// TIA Portal V16 export
// export: Created 2022-11-14T17:35:26.3349188Z, ExportSetting WithDefaults, DisplayName Totally Integrated Automation Portal, DisplayVersion V16, DisplayName TIA Portal Version Control Interface, DisplayVersion V16, DisplayName TIA Portal Openness, DisplayVersion V16, DisplayName STEP 7 Professional, DisplayVersion V16, DisplayName STEP 7 Safety, DisplayVersion V16, DisplayName WinCC Advanced, DisplayVersion V16
FUNCTION "FC32_ConveyorInverter_REV" : Void   // FC32, LAD
TITLE = Conveyor management with inverter
{ S7_Optimized_Access := 'FALSE' }
AUTHOR : Robopac
VERSION : 0.0
// stored: AutoNumber false, IsIECCheckEnabled false, SetENOAutomatically false, UDAEnableTagReadback false
   VAR_TEMP
      TimeUpwardTableCycle : Word;
      TimeUpwardTableCycleInt : Int;
      TempWord : Word;
   END_VAR
   VAR_TEMP   // added for the SCL form of the ladder/FBD networks
      _w1 : Bool;
   END_VAR
BEGIN

REGION Network 1: Timer SA type for conveyor motor
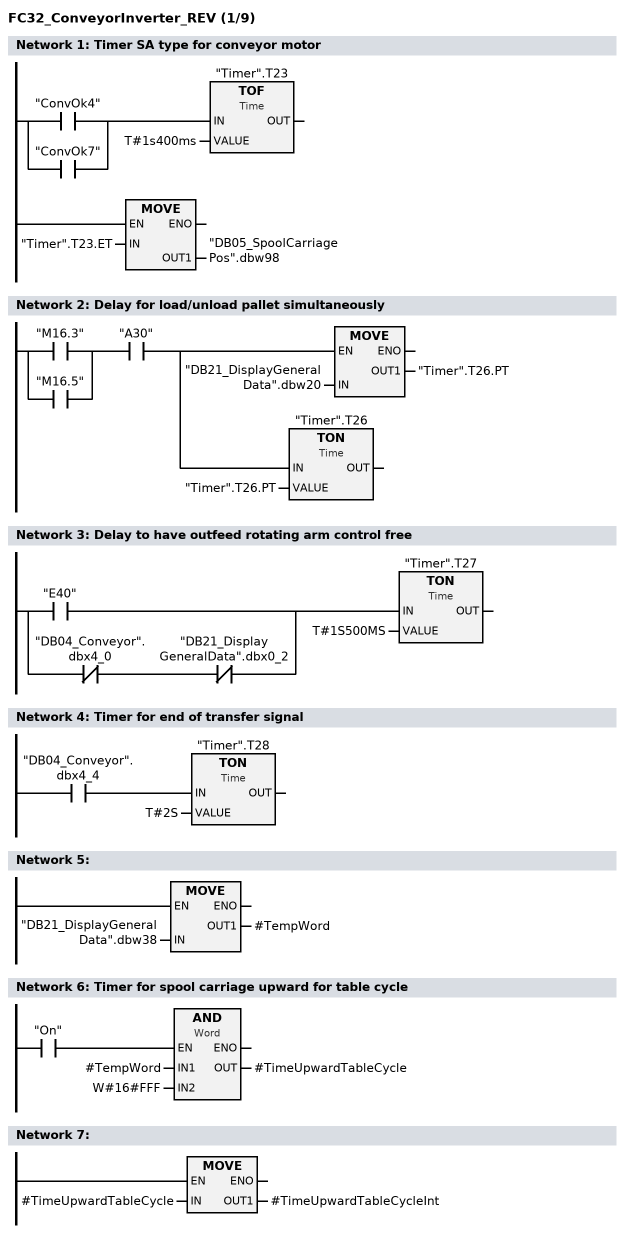
   "Timer".T23.TOF(IN := "ConvOk4" OR "ConvOk7", PT := T#1s400ms);   // TOF coil
   "DB05_SpoolCarriagePos".dbw98 := "Timer".T23.ET;
END_REGION

REGION Network 2: Delay for load/unload pallet simultaneously
   #_w1 := ("M16.3" OR "M16.5") AND "A30";
   IF #_w1 THEN "Timer".T26.PT := "DB21_DisplayGeneralData".dbw20; END_IF;
   "Timer".T26.TON(IN := #_w1, PT := "Timer".T26.PT);   // TON coil
END_REGION

REGION Network 3: Delay to have outfeed rotating arm control free
   "Timer".T27.TON(IN := "E40" OR (NOT "DB04_Conveyor".dbx4_0 AND NOT "DB21_DisplayGeneralData".dbx0_2), PT := T#1S500MS);   // TON coil
END_REGION

REGION Network 4: Timer for end of transfer signal
   "Timer".T28.TON(IN := "DB04_Conveyor".dbx4_4, PT := T#2S);   // TON coil
END_REGION

REGION Network 5
   RUNG wire#powerrail
      { S7_GenerateENO := "TRUE" } Move(in := "DB21_DisplayGeneralData".dbw38, out1 => #TempWord)
   END_RUNG
   // the same network as SCL:
   #TempWord := "DB21_DisplayGeneralData".dbw38;
END_REGION

REGION Network 6: Timer for spool carriage upward for table cycle
   RUNG wire#powerrail
      Contact( "On" )
      { S7_Templates := "SrcType := Word"; S7_GenerateENO := "TRUE" } And(in1 := #TempWord, in2 := W#16#FFF, out => #TimeUpwardTableCycle)
   END_RUNG
   // the same network as SCL:
   IF "On" THEN #TimeUpwardTableCycle := #TempWord AND W#16#FFF; END_IF;
END_REGION

REGION Network 7
   RUNG wire#powerrail
      { S7_GenerateENO := "TRUE" } Move(in := #TimeUpwardTableCycle, out1 => #TimeUpwardTableCycleInt)
   END_RUNG
   // the same network as SCL:
   #TimeUpwardTableCycleInt := #TimeUpwardTableCycle;
END_REGION

REGION Network 8: Timer for spool carriage upward for table cycle
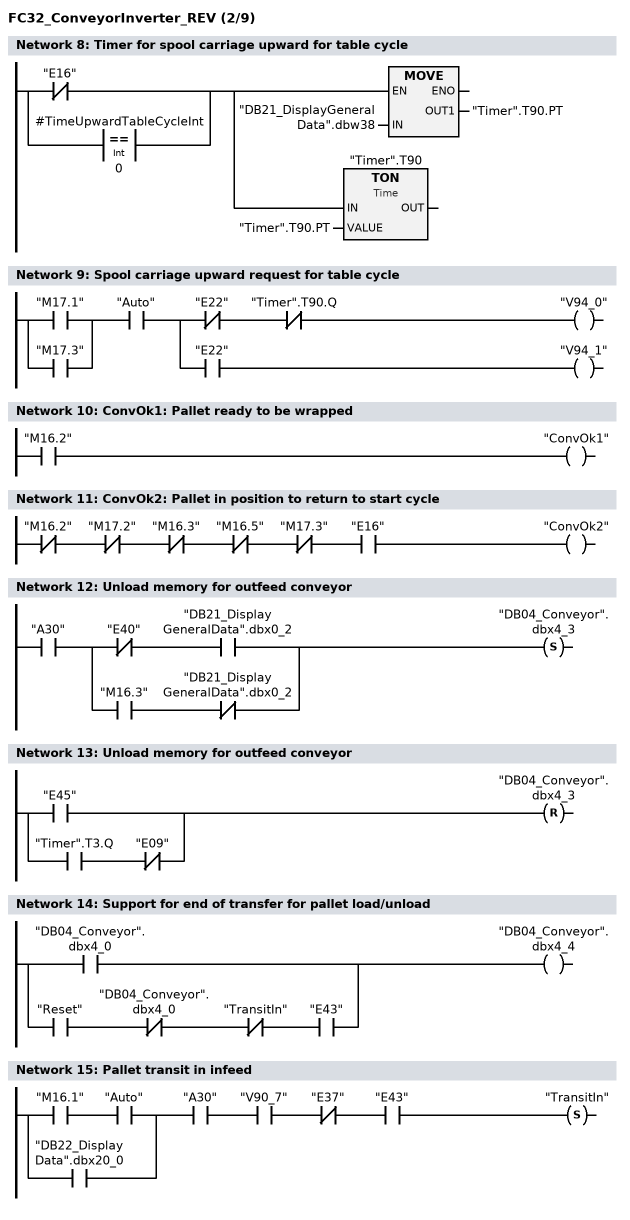
   #_w1 := NOT "E16" OR (#TimeUpwardTableCycleInt = 0);
   IF #_w1 THEN "Timer".T90.PT := "DB21_DisplayGeneralData".dbw38; END_IF;
   "Timer".T90.TON(IN := #_w1, PT := "Timer".T90.PT);   // TON coil
END_REGION

REGION Network 9: Spool carriage upward request for table cycle
   RUNG wire#powerrail
      Contact( "M17.1" )
      wire#w1
      Contact( "Auto" )
      wire#w2
      I_Contact( "E22" )
      I_Contact( "Timer".T90.Q )
      Coil( "V94_0" )
   END_RUNG
   RUNG wire#powerrail
      Contact( "M17.3" )
   END_RUNG wire#w1
   RUNG wire#w2
      Contact( "E22" )
      Coil( "V94_1" )
   END_RUNG
   // the same network as SCL:
   #_w1 := ("M17.1" OR "M17.3") AND "Auto";
   "V94_0" := #_w1 AND NOT "E22" AND NOT "Timer".T90.Q;
   "V94_1" := #_w1 AND "E22";
END_REGION

REGION Network 10: ConvOk1: Pallet ready to be wrapped
   RUNG wire#powerrail
      Contact( "M16.2" )
      Coil( "ConvOk1" )
   END_RUNG
   // the same network as SCL:
   "ConvOk1" := "M16.2";
END_REGION

REGION Network 11: ConvOk2: Pallet in position to return to start cycle
   RUNG wire#powerrail
      I_Contact( "M16.2" )
      I_Contact( "M17.2" )
      I_Contact( "M16.3" )
      I_Contact( "M16.5" )
      I_Contact( "M17.3" )
      Contact( "E16" )
      Coil( "ConvOk2" )
   END_RUNG
   // the same network as SCL:
   "ConvOk2" := NOT "M16.2" AND NOT "M17.2" AND NOT "M16.3" AND NOT "M16.5" AND NOT "M17.3" AND "E16";
END_REGION

REGION Network 12: Unload memory for outfeed conveyor
   RUNG wire#powerrail
      Contact( "A30" )
      wire#w1
      I_Contact( "E40" )
      Contact( "DB21_DisplayGeneralData".dbx0_2 )
      wire#w2
      S_Coil( "DB04_Conveyor".dbx4_3 )
   END_RUNG
   RUNG wire#w1
      Contact( "M16.3" )
      I_Contact( "DB21_DisplayGeneralData".dbx0_2 )
   END_RUNG wire#w2
   // the same network as SCL:
   IF "A30" AND ((NOT "E40" AND "DB21_DisplayGeneralData".dbx0_2) OR ("M16.3" AND NOT "DB21_DisplayGeneralData".dbx0_2)) THEN
       "DB04_Conveyor".dbx4_3 := TRUE;
   END_IF;
END_REGION

REGION Network 13: Unload memory for outfeed conveyor
   RUNG wire#powerrail
      Contact( "E45" )
      wire#w1
      R_Coil( "DB04_Conveyor".dbx4_3 )
   END_RUNG
   RUNG wire#powerrail
      Contact( "Timer".T3.Q )
      I_Contact( "E09" )
   END_RUNG wire#w1
   // the same network as SCL:
   IF "E45" OR ("Timer".T3.Q AND NOT "E09") THEN "DB04_Conveyor".dbx4_3 := FALSE; END_IF;
END_REGION

REGION Network 14: Support for end of transfer for pallet load/unload
   RUNG wire#powerrail
      Contact( "DB04_Conveyor".dbx4_0 )
      wire#w1
      Coil( "DB04_Conveyor".dbx4_4 )
   END_RUNG
   RUNG wire#powerrail
      Contact( "Reset" )
      I_Contact( "DB04_Conveyor".dbx4_0 )
      I_Contact( "TransitIn" )
      Contact( "E43" )
   END_RUNG wire#w1
   // the same network as SCL:
   "DB04_Conveyor".dbx4_4 := "DB04_Conveyor".dbx4_0 OR ("Reset" AND NOT "DB04_Conveyor".dbx4_0 AND NOT "TransitIn" AND "E43");
END_REGION

REGION Network 15: Pallet transit in infeed
   RUNG wire#powerrail
      Contact( "M16.1" )
      Contact( "Auto" )
      wire#w1
      Contact( "A30" )
      Contact( "V90_7" )
      I_Contact( "E37" )
      Contact( "E43" )
      S_Coil( "TransitIn" )
   END_RUNG
   RUNG wire#powerrail
      Contact( "DB22_DisplayData".dbx20_0 )
   END_RUNG wire#w1
   // the same network as SCL:
   IF (("M16.1" AND "Auto") OR "DB22_DisplayData".dbx20_0) AND "A30" AND "V90_7" AND NOT "E37" AND "E43" THEN
       "TransitIn" := TRUE;
   END_IF;
END_REGION

REGION Network 16: Pallet transit in infeed
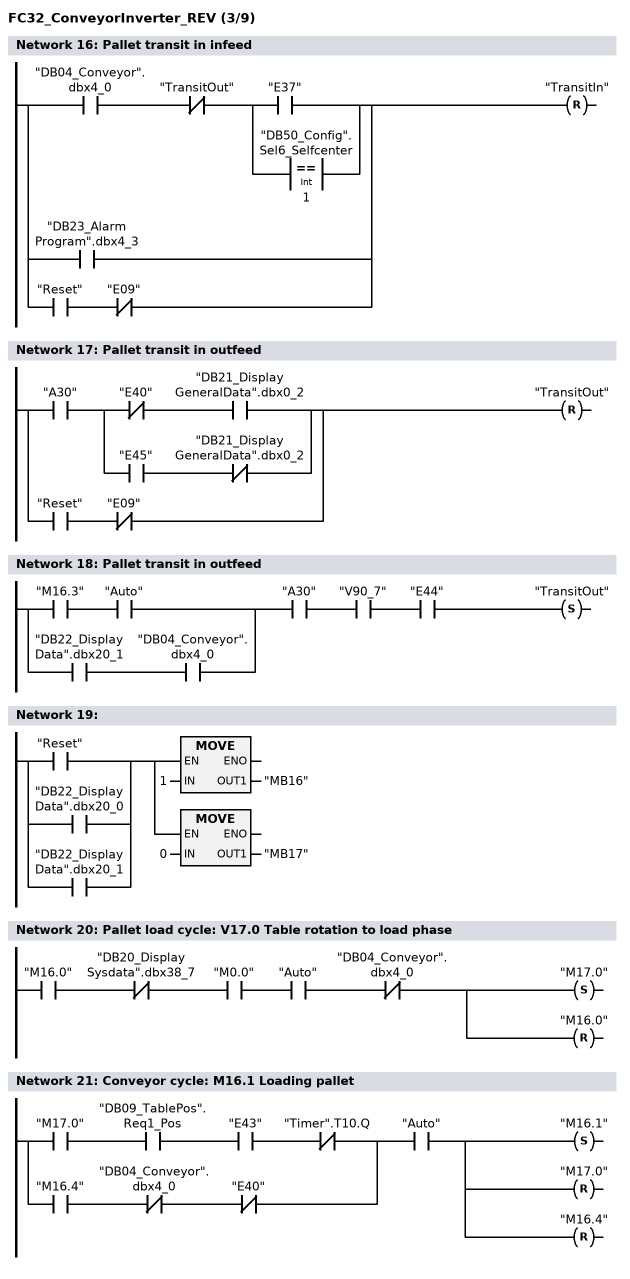
   IF ("DB04_Conveyor".dbx4_0 AND NOT "TransitOut" AND (("DB50_Config".Sel6_Selfcenter = 1) OR "E37")) OR "DB23_AlarmProgram".dbx4_3 OR ("Reset" AND NOT "E09") THEN
       "TransitIn" := FALSE;
   END_IF;
END_REGION

REGION Network 17: Pallet transit in outfeed
   RUNG wire#powerrail
      Contact( "A30" )
      wire#w1
      I_Contact( "E40" )
      Contact( "DB21_DisplayGeneralData".dbx0_2 )
      wire#w2
      R_Coil( "TransitOut" )
   END_RUNG
   RUNG wire#w1
      Contact( "E45" )
      I_Contact( "DB21_DisplayGeneralData".dbx0_2 )
   END_RUNG wire#w2
   RUNG wire#powerrail
      Contact( "Reset" )
      I_Contact( "E09" )
   END_RUNG wire#w2
   // the same network as SCL:
   IF ("A30" AND ((NOT "E40" AND "DB21_DisplayGeneralData".dbx0_2) OR ("E45" AND NOT "DB21_DisplayGeneralData".dbx0_2))) OR ("Reset" AND NOT "E09") THEN
       "TransitOut" := FALSE;
   END_IF;
END_REGION

REGION Network 18: Pallet transit in outfeed
   RUNG wire#powerrail
      Contact( "M16.3" )
      Contact( "Auto" )
      wire#w1
      Contact( "A30" )
      Contact( "V90_7" )
      Contact( "E44" )
      S_Coil( "TransitOut" )
   END_RUNG
   RUNG wire#powerrail
      Contact( "DB22_DisplayData".dbx20_1 )
      Contact( "DB04_Conveyor".dbx4_0 )
   END_RUNG wire#w1
   // the same network as SCL:
   IF (("M16.3" AND "Auto") OR ("DB22_DisplayData".dbx20_1 AND "DB04_Conveyor".dbx4_0)) AND "A30" AND "V90_7" AND "E44" THEN
       "TransitOut" := TRUE;
   END_IF;
END_REGION

REGION Network 19
   RUNG wire#powerrail
      Contact( "Reset" )
      wire#w1
      { S7_GenerateENO := "TRUE" } Move(in := 1, out1 => "MB16")
   END_RUNG
   RUNG wire#powerrail
      Contact( "DB22_DisplayData".dbx20_0 )
   END_RUNG wire#w1
   RUNG wire#powerrail
      Contact( "DB22_DisplayData".dbx20_1 )
   END_RUNG wire#w1
   RUNG wire#w1
      { S7_GenerateENO := "TRUE" } Move(in := 0, out1 => "MB17")
   END_RUNG
   // the same network as SCL:
   IF "Reset" OR "DB22_DisplayData".dbx20_0 OR "DB22_DisplayData".dbx20_1 THEN
       "MB16" := 1;
       "MB17" := 0;
   END_IF;
END_REGION

REGION Network 20: Pallet load cycle: V17.0 Table rotation to load phase
   RUNG wire#powerrail
      Contact( "M16.0" )
      I_Contact( "DB20_DisplaySysdata".dbx38_7 )
      Contact( "M0.0" )
      Contact( "Auto" )
      I_Contact( "DB04_Conveyor".dbx4_0 )
      wire#w1
      S_Coil( "M17.0" )
   END_RUNG
   RUNG wire#w1
      R_Coil( "M16.0" )
   END_RUNG
   // the same network as SCL:
   IF "M16.0" AND NOT "DB20_DisplaySysdata".dbx38_7 AND "M0.0" AND "Auto" AND NOT "DB04_Conveyor".dbx4_0 THEN
       "M17.0" := TRUE;
       "M16.0" := FALSE;
   END_IF;
END_REGION

REGION Network 21: Conveyor cycle: M16.1 Loading pallet
   RUNG wire#powerrail
      Contact( "M17.0" )
      Contact( "DB09_TablePos".Req1_Pos )
      Contact( "E43" )
      I_Contact( "Timer".T10.Q )
      wire#w1
      Contact( "Auto" )
      wire#w2
      S_Coil( "M16.1" )
   END_RUNG
   RUNG wire#powerrail
      Contact( "M16.4" )
      I_Contact( "DB04_Conveyor".dbx4_0 )
      I_Contact( "E40" )
   END_RUNG wire#w1
   RUNG wire#w2
      R_Coil( "M17.0" )
   END_RUNG
   RUNG wire#w2
      R_Coil( "M16.4" )
   END_RUNG
   // the same network as SCL:
   IF (("M17.0" AND "DB09_TablePos".Req1_Pos AND "E43" AND NOT "Timer".T10.Q) OR ("M16.4" AND NOT "DB04_Conveyor".dbx4_0 AND NOT "E40")) AND "Auto" THEN
       "M16.1" := TRUE;
   END_IF;
   #_w1 := (("M17.0" AND "DB09_TablePos".Req1_Pos AND "E43" AND NOT "Timer".T10.Q) OR ("M16.4" AND NOT "DB04_Conveyor".dbx4_0 AND NOT "E40")) AND "Auto";
   IF #_w1 THEN
       "M17.0" := FALSE;
       "M16.4" := FALSE;
   END_IF;
END_REGION

REGION Network 22: Pallet load cycle: V17.1 Table rotation to machine phase from lo
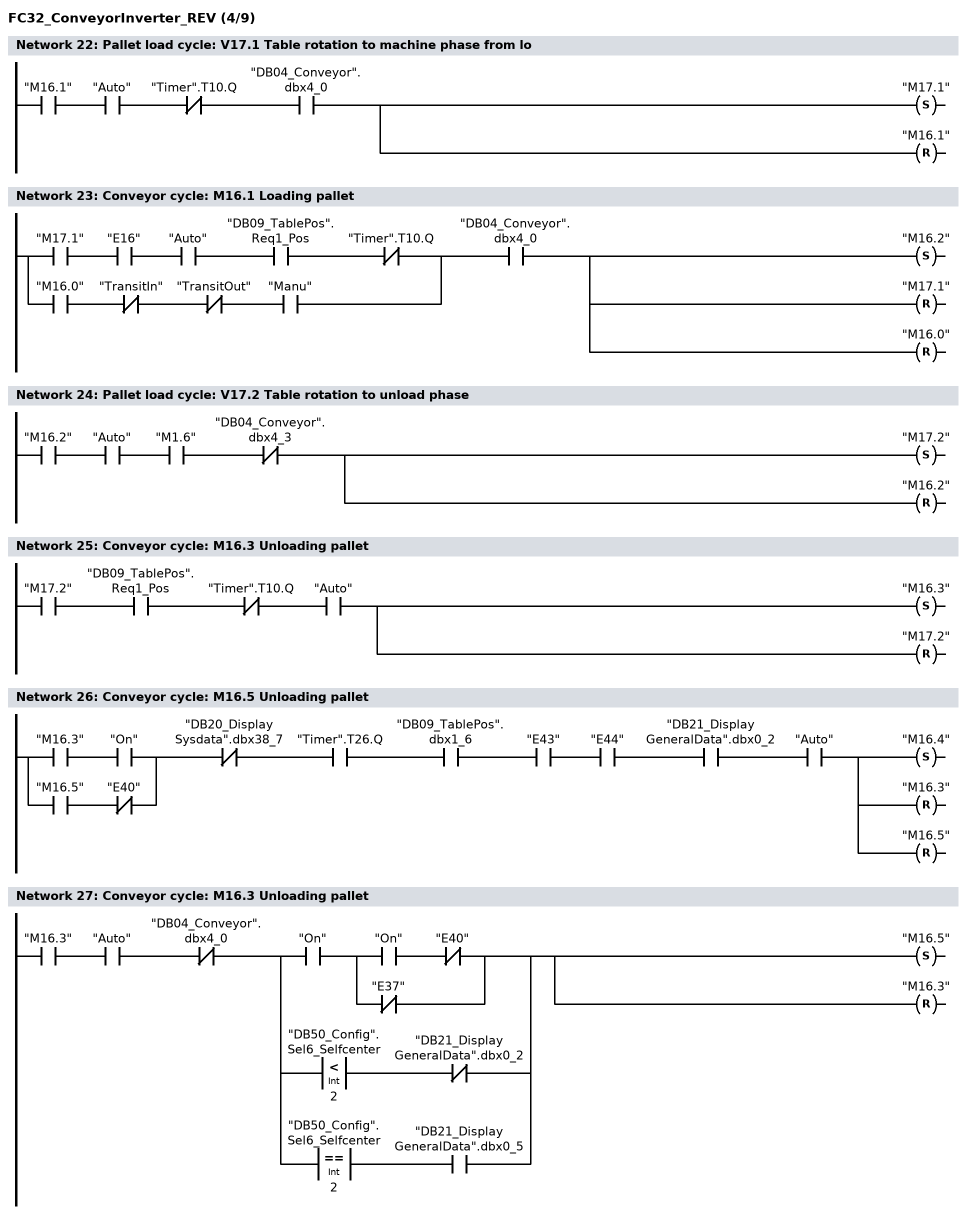
   RUNG wire#powerrail
      Contact( "M16.1" )
      Contact( "Auto" )
      I_Contact( "Timer".T10.Q )
      Contact( "DB04_Conveyor".dbx4_0 )
      wire#w1
      S_Coil( "M17.1" )
   END_RUNG
   RUNG wire#w1
      R_Coil( "M16.1" )
   END_RUNG
   // the same network as SCL:
   IF "M16.1" AND "Auto" AND NOT "Timer".T10.Q AND "DB04_Conveyor".dbx4_0 THEN
       "M17.1" := TRUE;
       "M16.1" := FALSE;
   END_IF;
END_REGION

REGION Network 23: Conveyor cycle: M16.1 Loading pallet
   RUNG wire#powerrail
      Contact( "M17.1" )
      Contact( "E16" )
      Contact( "Auto" )
      Contact( "DB09_TablePos".Req1_Pos )
      I_Contact( "Timer".T10.Q )
      wire#w1
      Contact( "DB04_Conveyor".dbx4_0 )
      wire#w2
      S_Coil( "M16.2" )
   END_RUNG
   RUNG wire#powerrail
      Contact( "M16.0" )
      I_Contact( "TransitIn" )
      I_Contact( "TransitOut" )
      Contact( "Manu" )
   END_RUNG wire#w1
   RUNG wire#w2
      R_Coil( "M17.1" )
   END_RUNG
   RUNG wire#w2
      R_Coil( "M16.0" )
   END_RUNG
   // the same network as SCL:
   IF (("M17.1" AND "E16" AND "Auto" AND "DB09_TablePos".Req1_Pos AND NOT "Timer".T10.Q) OR ("M16.0" AND NOT "TransitIn" AND NOT "TransitOut" AND "Manu")) AND "DB04_Conveyor".dbx4_0 THEN
       "M16.2" := TRUE;
   END_IF;
   #_w1 := (("M17.1" AND "E16" AND "Auto" AND "DB09_TablePos".Req1_Pos AND NOT "Timer".T10.Q) OR ("M16.0" AND NOT "TransitIn" AND NOT "TransitOut" AND "Manu")) AND "DB04_Conveyor".dbx4_0;
   IF #_w1 THEN
       "M17.1" := FALSE;
       "M16.0" := FALSE;
   END_IF;
END_REGION

REGION Network 24: Pallet load cycle: V17.2 Table rotation to unload phase
   RUNG wire#powerrail
      Contact( "M16.2" )
      Contact( "Auto" )
      Contact( "M1.6" )
      I_Contact( "DB04_Conveyor".dbx4_3 )
      wire#w1
      S_Coil( "M17.2" )
   END_RUNG
   RUNG wire#w1
      R_Coil( "M16.2" )
   END_RUNG
   // the same network as SCL:
   IF "M16.2" AND "Auto" AND "M1.6" AND NOT "DB04_Conveyor".dbx4_3 THEN
       "M17.2" := TRUE;
       "M16.2" := FALSE;
   END_IF;
END_REGION

REGION Network 25: Conveyor cycle: M16.3 Unloading pallet
   RUNG wire#powerrail
      Contact( "M17.2" )
      Contact( "DB09_TablePos".Req1_Pos )
      I_Contact( "Timer".T10.Q )
      Contact( "Auto" )
      wire#w1
      S_Coil( "M16.3" )
   END_RUNG
   RUNG wire#w1
      R_Coil( "M17.2" )
   END_RUNG
   // the same network as SCL:
   IF "M17.2" AND "DB09_TablePos".Req1_Pos AND NOT "Timer".T10.Q AND "Auto" THEN
       "M16.3" := TRUE;
       "M17.2" := FALSE;
   END_IF;
END_REGION

REGION Network 26: Conveyor cycle: M16.5 Unloading pallet
   RUNG wire#powerrail
      Contact( "M16.3" )
      Contact( "On" )
      wire#w1
      I_Contact( "DB20_DisplaySysdata".dbx38_7 )
      Contact( "Timer".T26.Q )
      Contact( "DB09_TablePos".dbx1_6 )
      Contact( "E43" )
      Contact( "E44" )
      Contact( "DB21_DisplayGeneralData".dbx0_2 )
      Contact( "Auto" )
      wire#w2
      S_Coil( "M16.4" )
   END_RUNG
   RUNG wire#powerrail
      Contact( "M16.5" )
      I_Contact( "E40" )
   END_RUNG wire#w1
   RUNG wire#w2
      R_Coil( "M16.3" )
   END_RUNG
   RUNG wire#w2
      R_Coil( "M16.5" )
   END_RUNG
   // the same network as SCL:
   IF (("M16.3" AND "On") OR ("M16.5" AND NOT "E40")) AND NOT "DB20_DisplaySysdata".dbx38_7 AND "Timer".T26.Q AND "DB09_TablePos".dbx1_6 AND "E43" AND "E44" AND "DB21_DisplayGeneralData".dbx0_2 AND "Auto" THEN
       "M16.4" := TRUE;
   END_IF;
   #_w1 := (("M16.3" AND "On") OR ("M16.5" AND NOT "E40")) AND NOT "DB20_DisplaySysdata".dbx38_7 AND "Timer".T26.Q AND "DB09_TablePos".dbx1_6 AND "E43" AND "E44" AND "DB21_DisplayGeneralData".dbx0_2 AND "Auto";
   IF #_w1 THEN
       "M16.3" := FALSE;
       "M16.5" := FALSE;
   END_IF;
END_REGION

REGION Network 27: Conveyor cycle: M16.3 Unloading pallet
   RUNG wire#powerrail
      Contact( "M16.3" )
      Contact( "Auto" )
      I_Contact( "DB04_Conveyor".dbx4_0 )
      wire#w1
      Contact( "On" )
      wire#w2
      Contact( "On" )
      I_Contact( "E40" )
      wire#w3
      S_Coil( "M16.5" )
   END_RUNG
   RUNG wire#w2
      I_Contact( "E37" )
   END_RUNG wire#w3
   RUNG wire#w1
      { S7_Templates := "SrcType := Int" } LT_Contact(in1 := "DB50_Config".Sel6_Selfcenter, in2 := 2)
      I_Contact( "DB21_DisplayGeneralData".dbx0_2 )
   END_RUNG wire#w3
   RUNG wire#w1
      { S7_Templates := "SrcType := Int" } EQ_Contact(in1 := "DB50_Config".Sel6_Selfcenter, in2 := 2)
      Contact( "DB21_DisplayGeneralData".dbx0_5 )
   END_RUNG wire#w3
   RUNG wire#w3
      R_Coil( "M16.3" )
   END_RUNG
   // the same network as SCL:
   IF "M16.3" AND "Auto" AND NOT "DB04_Conveyor".dbx4_0 AND (("On" AND (("On" AND NOT "E40") OR NOT "E37")) OR (("DB50_Config".Sel6_Selfcenter < 2) AND NOT "DB21_DisplayGeneralData".dbx0_2) OR (("DB50_Config".Sel6_Selfcenter = 2) AND "DB21_DisplayGeneralData".dbx0_5)) THEN
       "M16.5" := TRUE;
       "M16.3" := FALSE;
   END_IF;
END_REGION

REGION Network 28: Conveyor cycle: M16.5 Unloading pallet
   // CICLO FIERA
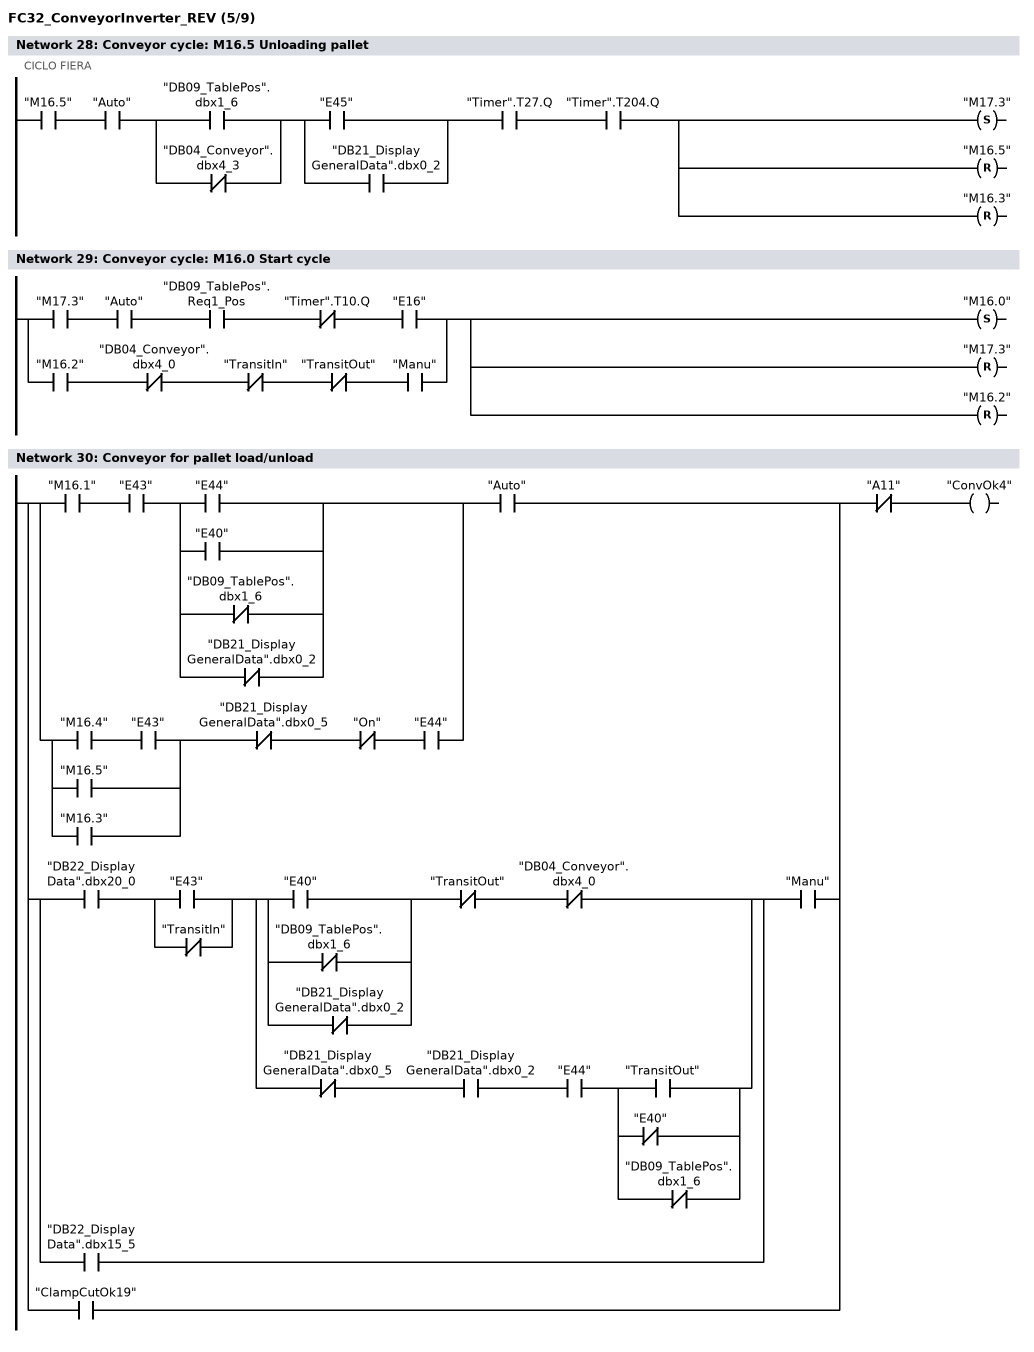
   RUNG wire#powerrail
      Contact( "M16.5" )
      Contact( "Auto" )
      wire#w1
      Contact( "DB09_TablePos".dbx1_6 )
      wire#w2
      Contact( "E45" )
      wire#w3
      Contact( "Timer".T27.Q )
      Contact( "Timer".T204.Q )
      wire#w4
      S_Coil( "M17.3" )
   END_RUNG
   RUNG wire#w1
      I_Contact( "DB04_Conveyor".dbx4_3 )
   END_RUNG wire#w2
   RUNG wire#w2
      Contact( "DB21_DisplayGeneralData".dbx0_2 )
   END_RUNG wire#w3
   RUNG wire#w4
      R_Coil( "M16.5" )
   END_RUNG
   RUNG wire#w4
      R_Coil( "M16.3" )
   END_RUNG
   // the same network as SCL:
   IF "M16.5" AND "Auto" AND ("DB09_TablePos".dbx1_6 OR NOT "DB04_Conveyor".dbx4_3) AND ("E45" OR "DB21_DisplayGeneralData".dbx0_2) AND "Timer".T27.Q AND "Timer".T204.Q THEN
       "M17.3" := TRUE;
   END_IF;
   #_w1 := "M16.5" AND "Auto" AND ("DB09_TablePos".dbx1_6 OR NOT "DB04_Conveyor".dbx4_3) AND ("E45" OR "DB21_DisplayGeneralData".dbx0_2) AND "Timer".T27.Q AND "Timer".T204.Q;
   IF #_w1 THEN
       "M16.5" := FALSE;
       "M16.3" := FALSE;
   END_IF;
END_REGION

REGION Network 29: Conveyor cycle: M16.0 Start cycle
   RUNG wire#powerrail
      Contact( "M17.3" )
      Contact( "Auto" )
      Contact( "DB09_TablePos".Req1_Pos )
      I_Contact( "Timer".T10.Q )
      Contact( "E16" )
      wire#w1
      S_Coil( "M16.0" )
   END_RUNG
   RUNG wire#powerrail
      Contact( "M16.2" )
      I_Contact( "DB04_Conveyor".dbx4_0 )
      I_Contact( "TransitIn" )
      I_Contact( "TransitOut" )
      Contact( "Manu" )
   END_RUNG wire#w1
   RUNG wire#w1
      R_Coil( "M17.3" )
   END_RUNG
   RUNG wire#w1
      R_Coil( "M16.2" )
   END_RUNG
   // the same network as SCL:
   IF ("M17.3" AND "Auto" AND "DB09_TablePos".Req1_Pos AND NOT "Timer".T10.Q AND "E16") OR ("M16.2" AND NOT "DB04_Conveyor".dbx4_0 AND NOT "TransitIn" AND NOT "TransitOut" AND "Manu") THEN
       "M16.0" := TRUE;
   END_IF;
   #_w1 := ("M17.3" AND "Auto" AND "DB09_TablePos".Req1_Pos AND NOT "Timer".T10.Q AND "E16") OR ("M16.2" AND NOT "DB04_Conveyor".dbx4_0 AND NOT "TransitIn" AND NOT "TransitOut" AND "Manu");
   IF #_w1 THEN
       "M17.3" := FALSE;
       "M16.2" := FALSE;
   END_IF;
END_REGION

REGION Network 30: Conveyor for pallet load/unload
   RUNG wire#powerrail
      Contact( "M16.1" )
      Contact( "E43" )
      wire#w1
      Contact( "E44" )
      wire#w2
      Contact( "Auto" )
      wire#w4
      I_Contact( "A11" )
      Coil( "ConvOk4" )
   END_RUNG
   RUNG wire#w1
      Contact( "E40" )
   END_RUNG wire#w2
   RUNG wire#w1
      I_Contact( "DB09_TablePos".dbx1_6 )
   END_RUNG wire#w2
   RUNG wire#w1
      I_Contact( "DB21_DisplayGeneralData".dbx0_2 )
   END_RUNG wire#w2
   RUNG wire#powerrail
      Contact( "M16.4" )
      Contact( "E43" )
      wire#w3
      I_Contact( "DB21_DisplayGeneralData".dbx0_5 )
      I_Contact( "On" )
      Contact( "E44" )
   END_RUNG wire#w2
   RUNG wire#powerrail
      Contact( "M16.5" )
   END_RUNG wire#w3
   RUNG wire#powerrail
      Contact( "M16.3" )
   END_RUNG wire#w3
   RUNG wire#powerrail
      Contact( "DB22_DisplayData".dbx20_0 )
      wire#w5
      Contact( "E43" )
      wire#w6
      Contact( "E40" )
      wire#w7
      I_Contact( "TransitOut" )
      I_Contact( "DB04_Conveyor".dbx4_0 )
      wire#w8
      Contact( "Manu" )
   END_RUNG wire#w4
   RUNG wire#w5
      I_Contact( "TransitIn" )
   END_RUNG wire#w6
   RUNG wire#w6
      I_Contact( "DB09_TablePos".dbx1_6 )
   END_RUNG wire#w7
   RUNG wire#w6
      I_Contact( "DB21_DisplayGeneralData".dbx0_2 )
   END_RUNG wire#w7
   RUNG wire#w6
      I_Contact( "DB21_DisplayGeneralData".dbx0_5 )
      Contact( "DB21_DisplayGeneralData".dbx0_2 )
      Contact( "E44" )
      wire#w9
      Contact( "TransitOut" )
   END_RUNG wire#w8
   RUNG wire#w9
      I_Contact( "E40" )
   END_RUNG wire#w8
   RUNG wire#w9
      I_Contact( "DB09_TablePos".dbx1_6 )
   END_RUNG wire#w8
   RUNG wire#powerrail
      Contact( "DB22_DisplayData".dbx15_5 )
   END_RUNG wire#w8
   RUNG wire#powerrail
      Contact( "ClampCutOk19" )
   END_RUNG wire#w4
   // the same network as SCL:
   "ConvOk4" := (((("M16.1" AND "E43" AND ("E44" OR "E40" OR NOT "DB09_TablePos".dbx1_6 OR NOT "DB21_DisplayGeneralData".dbx0_2)) OR ((("M16.4" AND "E43") OR "M16.5" OR "M16.3") AND NOT "DB21_DisplayGeneralData".dbx0_5 AND NOT "On" AND "E44")) AND "Auto") OR ((("DB22_DisplayData".dbx20_0 AND ("E43" OR NOT "TransitIn") AND ((("E40" OR NOT "DB09_TablePos".dbx1_6 OR NOT "DB21_DisplayGeneralData".dbx0_2) AND NOT "TransitOut" AND NOT "DB04_Conveyor".dbx4_0) OR (NOT "DB21_DisplayGeneralData".dbx0_5 AND "DB21_DisplayGeneralData".dbx0_2 AND "E44" AND ("TransitOut" OR NOT "E40" OR NOT "DB09_TablePos".dbx1_6)))) OR "DB22_DisplayData".dbx15_5) AND "Manu") OR "ClampCutOk19") AND NOT "A11";
END_REGION

REGION Network 31: ConvOk7: Backward for inverter
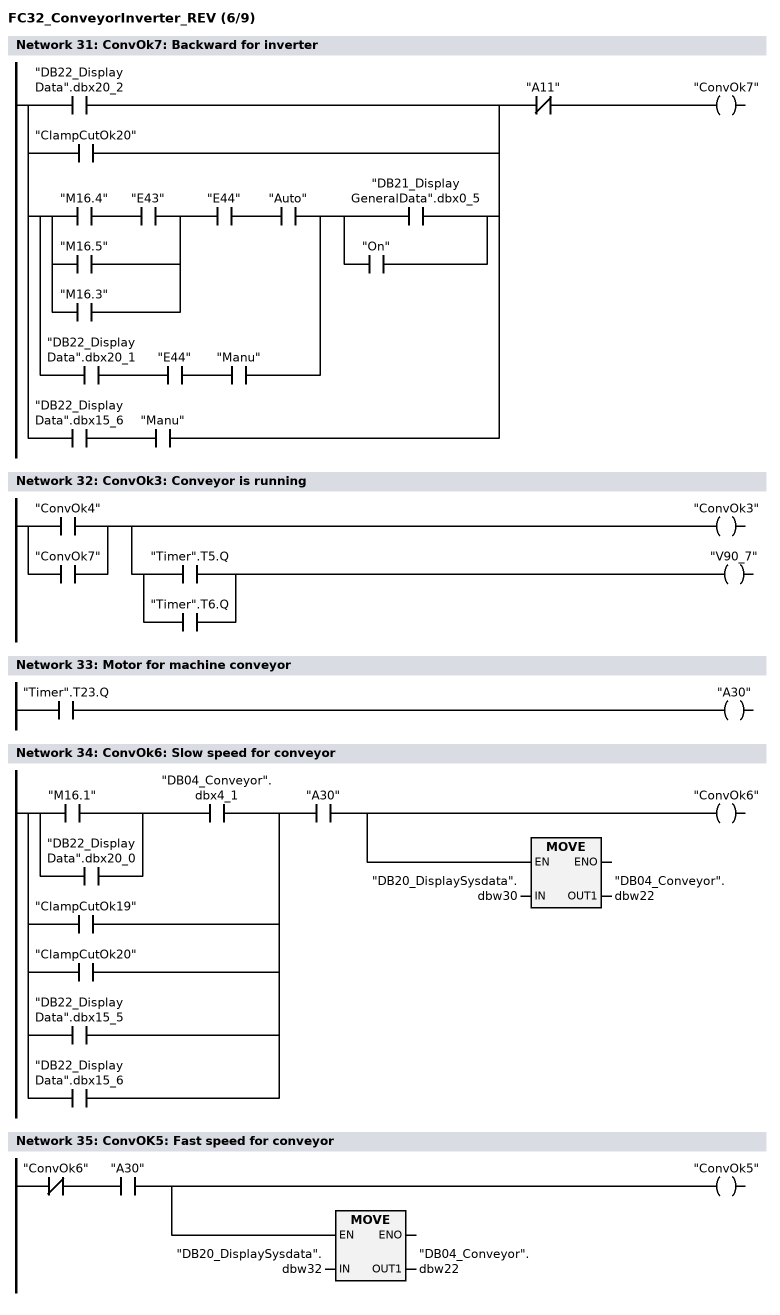
   RUNG wire#powerrail
      Contact( "DB22_DisplayData".dbx20_2 )
      wire#w1
      I_Contact( "A11" )
      Coil( "ConvOk7" )
   END_RUNG
   RUNG wire#powerrail
      Contact( "ClampCutOk20" )
   END_RUNG wire#w1
   RUNG wire#powerrail
      Contact( "M16.4" )
      Contact( "E43" )
      wire#w2
      Contact( "E44" )
      Contact( "Auto" )
      wire#w3
      Contact( "DB21_DisplayGeneralData".dbx0_5 )
   END_RUNG wire#w1
   RUNG wire#powerrail
      Contact( "M16.5" )
   END_RUNG wire#w2
   RUNG wire#powerrail
      Contact( "M16.3" )
   END_RUNG wire#w2
   RUNG wire#powerrail
      Contact( "DB22_DisplayData".dbx20_1 )
      Contact( "E44" )
      Contact( "Manu" )
   END_RUNG wire#w3
   RUNG wire#w3
      Contact( "On" )
   END_RUNG wire#w1
   RUNG wire#powerrail
      Contact( "DB22_DisplayData".dbx15_6 )
      Contact( "Manu" )
   END_RUNG wire#w1
   // the same network as SCL:
   "ConvOk7" := ("DB22_DisplayData".dbx20_2 OR "ClampCutOk20" OR ((((("M16.4" AND "E43") OR "M16.5" OR "M16.3") AND "E44" AND "Auto") OR ("DB22_DisplayData".dbx20_1 AND "E44" AND "Manu")) AND ("DB21_DisplayGeneralData".dbx0_5 OR "On")) OR ("DB22_DisplayData".dbx15_6 AND "Manu")) AND NOT "A11";
END_REGION

REGION Network 32: ConvOk3: Conveyor is running
   RUNG wire#powerrail
      Contact( "ConvOk4" )
      wire#w1
      Coil( "ConvOk3" )
   END_RUNG
   RUNG wire#powerrail
      Contact( "ConvOk7" )
   END_RUNG wire#w1
   RUNG wire#w1
      Contact( "Timer".T5.Q )
      wire#w2
      Coil( "V90_7" )
   END_RUNG
   RUNG wire#w1
      Contact( "Timer".T6.Q )
   END_RUNG wire#w2
   // the same network as SCL:
   "ConvOk3" := "ConvOk4" OR "ConvOk7";
   "V90_7" := "ConvOk3" AND ("Timer".T5.Q OR "Timer".T6.Q);
END_REGION

REGION Network 33: Motor for machine conveyor
   RUNG wire#powerrail
      Contact( "Timer".T23.Q )
      Coil( "A30" )
   END_RUNG
   // the same network as SCL:
   "A30" := "Timer".T23.Q;
END_REGION

REGION Network 34: ConvOk6: Slow speed for conveyor
   RUNG wire#powerrail
      Contact( "M16.1" )
      wire#w1
      Contact( "DB04_Conveyor".dbx4_1 )
      wire#w2
      Contact( "A30" )
      wire#w3
      Coil( "ConvOk6" )
   END_RUNG
   RUNG wire#powerrail
      Contact( "DB22_DisplayData".dbx20_0 )
   END_RUNG wire#w1
   RUNG wire#powerrail
      Contact( "ClampCutOk19" )
   END_RUNG wire#w2
   RUNG wire#powerrail
      Contact( "ClampCutOk20" )
   END_RUNG wire#w2
   RUNG wire#powerrail
      Contact( "DB22_DisplayData".dbx15_5 )
   END_RUNG wire#w2
   RUNG wire#powerrail
      Contact( "DB22_DisplayData".dbx15_6 )
   END_RUNG wire#w2
   RUNG wire#w3
      { S7_GenerateENO := "TRUE" } Move(in := "DB20_DisplaySysdata".dbw30, out1 => "DB04_Conveyor".dbw22)
   END_RUNG
   // the same network as SCL:
   "ConvOk6" := ((("M16.1" OR "DB22_DisplayData".dbx20_0) AND "DB04_Conveyor".dbx4_1) OR "ClampCutOk19" OR "ClampCutOk20" OR "DB22_DisplayData".dbx15_5 OR "DB22_DisplayData".dbx15_6) AND "A30";
   IF "ConvOk6" THEN "DB04_Conveyor".dbw22 := "DB20_DisplaySysdata".dbw30; END_IF;
END_REGION

REGION Network 35: ConvOK5: Fast speed for conveyor
   RUNG wire#powerrail
      I_Contact( "ConvOk6" )
      Contact( "A30" )
      wire#w1
      Coil( "ConvOk5" )
   END_RUNG
   RUNG wire#w1
      { S7_GenerateENO := "TRUE" } Move(in := "DB20_DisplaySysdata".dbw32, out1 => "DB04_Conveyor".dbw22)
   END_RUNG
   // the same network as SCL:
   "ConvOk5" := NOT "ConvOk6" AND "A30";
   IF "ConvOk5" THEN "DB04_Conveyor".dbw22 := "DB20_DisplaySysdata".dbw32; END_IF;
END_REGION

REGION Network 36: rotation inverter: Support for speed selection
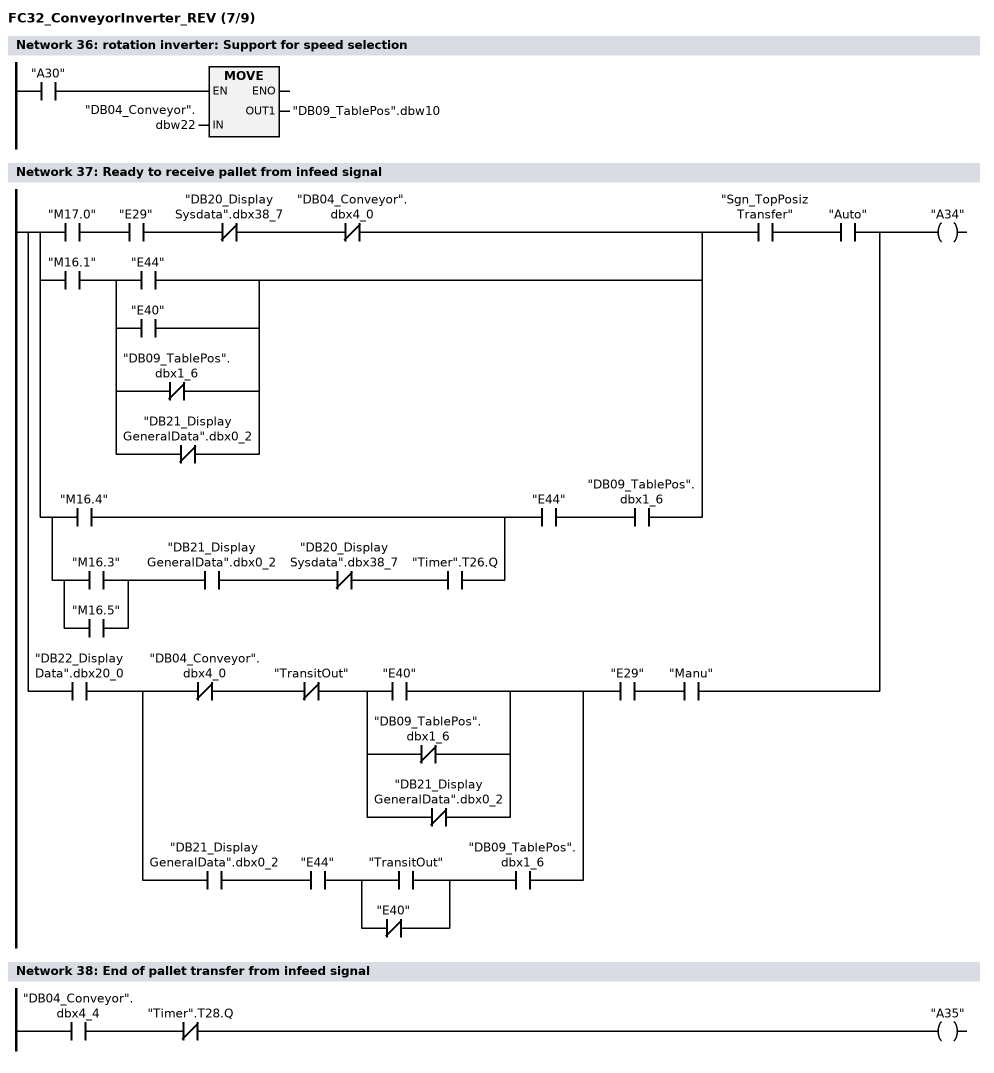
   RUNG wire#powerrail
      Contact( "A30" )
      { S7_GenerateENO := "TRUE" } Move(in := "DB04_Conveyor".dbw22, out1 => "DB09_TablePos".dbw10)
   END_RUNG
   // the same network as SCL:
   IF "A30" THEN "DB09_TablePos".dbw10 := "DB04_Conveyor".dbw22; END_IF;
END_REGION

REGION Network 37: Ready to receive pallet from infeed signal
   RUNG wire#powerrail
      Contact( "M17.0" )
      Contact( "E29" )
      I_Contact( "DB20_DisplaySysdata".dbx38_7 )
      I_Contact( "DB04_Conveyor".dbx4_0 )
      wire#w1
      Contact( "Sgn_TopPosizTransfer" )
      Contact( "Auto" )
      wire#w5
      Coil( "A34" )
   END_RUNG
   RUNG wire#powerrail
      Contact( "M16.1" )
      wire#w2
      Contact( "E44" )
   END_RUNG wire#w1
   RUNG wire#w2
      Contact( "E40" )
   END_RUNG wire#w1
   RUNG wire#w2
      I_Contact( "DB09_TablePos".dbx1_6 )
   END_RUNG wire#w1
   RUNG wire#w2
      I_Contact( "DB21_DisplayGeneralData".dbx0_2 )
   END_RUNG wire#w1
   RUNG wire#powerrail
      Contact( "M16.4" )
      wire#w3
      Contact( "E44" )
      Contact( "DB09_TablePos".dbx1_6 )
   END_RUNG wire#w1
   RUNG wire#powerrail
      Contact( "M16.3" )
      wire#w4
      Contact( "DB21_DisplayGeneralData".dbx0_2 )
      I_Contact( "DB20_DisplaySysdata".dbx38_7 )
      Contact( "Timer".T26.Q )
   END_RUNG wire#w3
   RUNG wire#powerrail
      Contact( "M16.5" )
   END_RUNG wire#w4
   RUNG wire#powerrail
      Contact( "DB22_DisplayData".dbx20_0 )
      wire#w6
      I_Contact( "DB04_Conveyor".dbx4_0 )
      I_Contact( "TransitOut" )
      wire#w7
      Contact( "E40" )
      wire#w8
      Contact( "E29" )
      Contact( "Manu" )
   END_RUNG wire#w5
   RUNG wire#w7
      I_Contact( "DB09_TablePos".dbx1_6 )
   END_RUNG wire#w8
   RUNG wire#w7
      I_Contact( "DB21_DisplayGeneralData".dbx0_2 )
   END_RUNG wire#w8
   RUNG wire#w6
      Contact( "DB21_DisplayGeneralData".dbx0_2 )
      Contact( "E44" )
      wire#w9
      Contact( "TransitOut" )
      wire#w10
      Contact( "DB09_TablePos".dbx1_6 )
   END_RUNG wire#w8
   RUNG wire#w9
      I_Contact( "E40" )
   END_RUNG wire#w10
   // the same network as SCL:
   "A34" := ((("M17.0" AND "E29" AND NOT "DB20_DisplaySysdata".dbx38_7 AND NOT "DB04_Conveyor".dbx4_0) OR ("M16.1" AND ("E44" OR "E40" OR NOT "DB09_TablePos".dbx1_6 OR NOT "DB21_DisplayGeneralData".dbx0_2)) OR (("M16.4" OR (("M16.3" OR "M16.5") AND "DB21_DisplayGeneralData".dbx0_2 AND NOT "DB20_DisplaySysdata".dbx38_7 AND "Timer".T26.Q)) AND "E44" AND "DB09_TablePos".dbx1_6)) AND "Sgn_TopPosizTransfer" AND "Auto") OR ("DB22_DisplayData".dbx20_0 AND ((NOT "DB04_Conveyor".dbx4_0 AND NOT "TransitOut" AND ("E40" OR NOT "DB09_TablePos".dbx1_6 OR NOT "DB21_DisplayGeneralData".dbx0_2)) OR ("DB21_DisplayGeneralData".dbx0_2 AND "E44" AND ("TransitOut" OR NOT "E40") AND "DB09_TablePos".dbx1_6)) AND "E29" AND "Manu");
END_REGION

REGION Network 38: End of pallet transfer from infeed signal
   RUNG wire#powerrail
      Contact( "DB04_Conveyor".dbx4_4 )
      I_Contact( "Timer".T28.Q )
      Coil( "A35" )
   END_RUNG
   // the same network as SCL:
   "A35" := "DB04_Conveyor".dbx4_4 AND NOT "Timer".T28.Q;
END_REGION

REGION Network 39: Pallet ready for outfeed signal
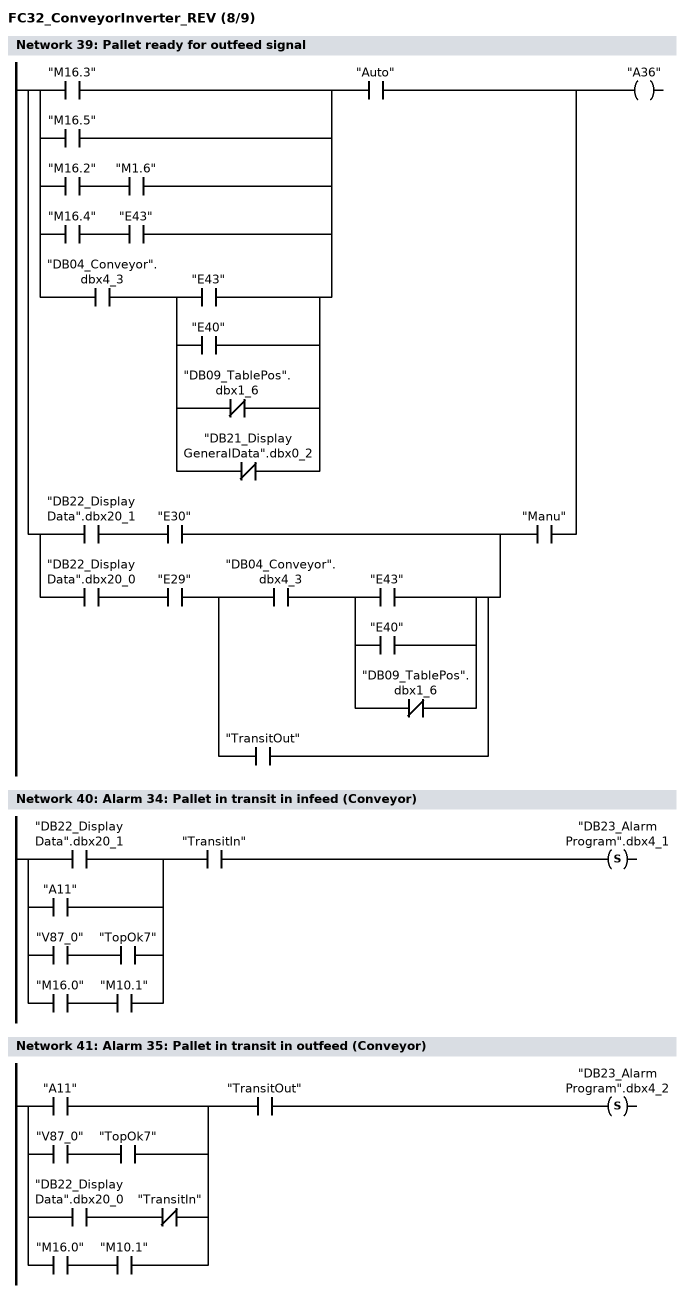
   RUNG wire#powerrail
      Contact( "M16.3" )
      wire#w1
      Contact( "Auto" )
      wire#w3
      Coil( "A36" )
   END_RUNG
   RUNG wire#powerrail
      Contact( "M16.5" )
   END_RUNG wire#w1
   RUNG wire#powerrail
      Contact( "M16.2" )
      Contact( "M1.6" )
   END_RUNG wire#w1
   RUNG wire#powerrail
      Contact( "M16.4" )
      Contact( "E43" )
   END_RUNG wire#w1
   RUNG wire#powerrail
      Contact( "DB04_Conveyor".dbx4_3 )
      wire#w2
      Contact( "E43" )
   END_RUNG wire#w1
   RUNG wire#w2
      Contact( "E40" )
   END_RUNG wire#w1
   RUNG wire#w2
      I_Contact( "DB09_TablePos".dbx1_6 )
   END_RUNG wire#w1
   RUNG wire#w2
      I_Contact( "DB21_DisplayGeneralData".dbx0_2 )
   END_RUNG wire#w1
   RUNG wire#powerrail
      Contact( "DB22_DisplayData".dbx20_1 )
      Contact( "E30" )
      wire#w4
      Contact( "Manu" )
   END_RUNG wire#w3
   RUNG wire#powerrail
      Contact( "DB22_DisplayData".dbx20_0 )
      Contact( "E29" )
      wire#w5
      Contact( "DB04_Conveyor".dbx4_3 )
      wire#w6
      Contact( "E43" )
   END_RUNG wire#w4
   RUNG wire#w6
      Contact( "E40" )
   END_RUNG wire#w4
   RUNG wire#w6
      I_Contact( "DB09_TablePos".dbx1_6 )
   END_RUNG wire#w4
   RUNG wire#w5
      Contact( "TransitOut" )
   END_RUNG wire#w4
   // the same network as SCL:
   "A36" := (("M16.3" OR "M16.5" OR ("M16.2" AND "M1.6") OR ("M16.4" AND "E43") OR ("DB04_Conveyor".dbx4_3 AND ("E43" OR "E40" OR NOT "DB09_TablePos".dbx1_6 OR NOT "DB21_DisplayGeneralData".dbx0_2))) AND "Auto") OR ((("DB22_DisplayData".dbx20_1 AND "E30") OR ("DB22_DisplayData".dbx20_0 AND "E29" AND (("DB04_Conveyor".dbx4_3 AND ("E43" OR "E40" OR NOT "DB09_TablePos".dbx1_6)) OR "TransitOut"))) AND "Manu");
END_REGION

REGION Network 40: Alarm 34: Pallet in transit in infeed (Conveyor)
   RUNG wire#powerrail
      Contact( "DB22_DisplayData".dbx20_1 )
      wire#w1
      Contact( "TransitIn" )
      S_Coil( "DB23_AlarmProgram".dbx4_1 )
   END_RUNG
   RUNG wire#powerrail
      Contact( "A11" )
   END_RUNG wire#w1
   RUNG wire#powerrail
      Contact( "V87_0" )
      Contact( "TopOk7" )
   END_RUNG wire#w1
   RUNG wire#powerrail
      Contact( "M16.0" )
      Contact( "M10.1" )
   END_RUNG wire#w1
   // the same network as SCL:
   IF ("DB22_DisplayData".dbx20_1 OR "A11" OR ("V87_0" AND "TopOk7") OR ("M16.0" AND "M10.1")) AND "TransitIn" THEN
       "DB23_AlarmProgram".dbx4_1 := TRUE;
   END_IF;
END_REGION

REGION Network 41: Alarm 35: Pallet in transit in outfeed (Conveyor)
   RUNG wire#powerrail
      Contact( "A11" )
      wire#w1
      Contact( "TransitOut" )
      S_Coil( "DB23_AlarmProgram".dbx4_2 )
   END_RUNG
   RUNG wire#powerrail
      Contact( "V87_0" )
      Contact( "TopOk7" )
   END_RUNG wire#w1
   RUNG wire#powerrail
      Contact( "DB22_DisplayData".dbx20_0 )
      I_Contact( "TransitIn" )
   END_RUNG wire#w1
   RUNG wire#powerrail
      Contact( "M16.0" )
      Contact( "M10.1" )
   END_RUNG wire#w1
   // the same network as SCL:
   IF ("A11" OR ("V87_0" AND "TopOk7") OR ("DB22_DisplayData".dbx20_0 AND NOT "TransitIn") OR ("M16.0" AND "M10.1")) AND "TransitOut" THEN
       "DB23_AlarmProgram".dbx4_2 := TRUE;
   END_IF;
END_REGION

REGION Network 42: Alarm 39: Technoplat table not in load phase
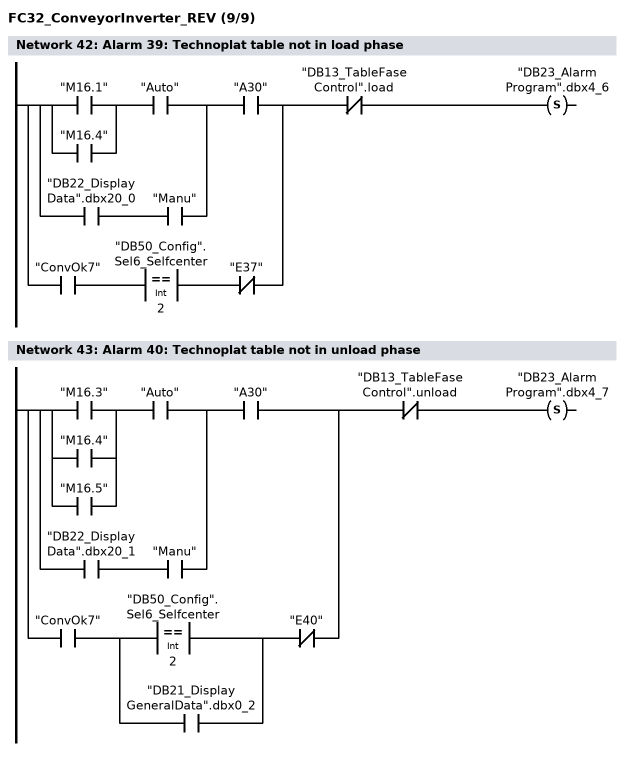
   RUNG wire#powerrail
      Contact( "M16.1" )
      wire#w1
      Contact( "Auto" )
      wire#w2
      Contact( "A30" )
      wire#w3
      I_Contact( "DB13_TableFaseControl".load )
      S_Coil( "DB23_AlarmProgram".dbx4_6 )
   END_RUNG
   RUNG wire#powerrail
      Contact( "M16.4" )
   END_RUNG wire#w1
   RUNG wire#powerrail
      Contact( "DB22_DisplayData".dbx20_0 )
      Contact( "Manu" )
   END_RUNG wire#w2
   RUNG wire#powerrail
      Contact( "ConvOk7" )
      { S7_Templates := "SrcType := Int" } EQ_Contact(in1 := "DB50_Config".Sel6_Selfcenter, in2 := 2)
      I_Contact( "E37" )
   END_RUNG wire#w3
   // the same network as SCL:
   IF ((((("M16.1" OR "M16.4") AND "Auto") OR ("DB22_DisplayData".dbx20_0 AND "Manu")) AND "A30") OR ("ConvOk7" AND ("DB50_Config".Sel6_Selfcenter = 2) AND NOT "E37")) AND NOT "DB13_TableFaseControl".load THEN
       "DB23_AlarmProgram".dbx4_6 := TRUE;
   END_IF;
END_REGION

REGION Network 43: Alarm 40: Technoplat table not in unload phase
   RUNG wire#powerrail
      Contact( "M16.3" )
      wire#w1
      Contact( "Auto" )
      wire#w2
      Contact( "A30" )
      wire#w3
      I_Contact( "DB13_TableFaseControl".unload )
      S_Coil( "DB23_AlarmProgram".dbx4_7 )
   END_RUNG
   RUNG wire#powerrail
      Contact( "M16.4" )
   END_RUNG wire#w1
   RUNG wire#powerrail
      Contact( "M16.5" )
   END_RUNG wire#w1
   RUNG wire#powerrail
      Contact( "DB22_DisplayData".dbx20_1 )
      Contact( "Manu" )
   END_RUNG wire#w2
   RUNG wire#powerrail
      Contact( "ConvOk7" )
      wire#w4
      { S7_Templates := "SrcType := Int" } EQ_Contact(in1 := "DB50_Config".Sel6_Selfcenter, in2 := 2)
      wire#w5
      I_Contact( "E40" )
   END_RUNG wire#w3
   RUNG wire#w4
      Contact( "DB21_DisplayGeneralData".dbx0_2 )
   END_RUNG wire#w5
   // the same network as SCL:
   IF ((((("M16.3" OR "M16.4" OR "M16.5") AND "Auto") OR ("DB22_DisplayData".dbx20_1 AND "Manu")) AND "A30") OR ("ConvOk7" AND (("DB50_Config".Sel6_Selfcenter = 2) OR "DB21_DisplayGeneralData".dbx0_2) AND NOT "E40")) AND NOT "DB13_TableFaseControl".unload THEN
       "DB23_AlarmProgram".dbx4_7 := TRUE;
   END_IF;
END_REGION
END_FUNCTION
